FUNCTION_BLOCK Derivative_Tests EXTENDS FB_TestSuite
VAR
    delta : LREAL := 1e-5;
END_VAR

FirstCallDerivateiveIsZero();
CalculatederivateOnSecondCall();

METHOD CalculatederivateOnSecondCall
VAR_INST
    d : Derivative;
END_VAR
TEST('CalculatederivateOnSecondCall');

d(value:=1, deltatime:=1);
d(value:=2, deltatime:=1);

AssertEquals_LREAL(Expected:=1, Actual:=d.Out, Delta:=delta, Message:='derivative not correct');

TcUnit.TEST_FINISHED();
END_METHOD

METHOD FirstCallDerivateiveIsZero
VAR_INST
    d : Derivative;
END_VAR
TEST('FirstCallDerivateiveIsZero');

d(value:=1, deltatime:=1);

AssertEquals_LREAL(Expected:=0, Actual:=d.Out, Delta:=delta, Message:='derivative not correct');

TcUnit.TEST_FINISHED();
END_METHOD

END_FUNCTION_BLOCK

(* stored: Version 1.1.0.1, ProductVersion 3.1.4024.12
   POU Derivative_Tests: Id {139527eb-4a04-441d-876d-9180e432d73f}, SpecialFunc None
   Method CalculatederivateOnSecondCall: Id {5ea7d5fb-18e0-44e8-b58f-e05af34347f1}
   Method FirstCallDerivateiveIsZero: Id {7d6d5b14-8a46-4c91-ad29-b972df5220ba} *)
